FUNCTION_BLOCK FB_AlarmDelay
VAR_INPUT
	msec				: INT;
	alarmState			: BOOL;
	alarmResetTimer		: BOOL;
END_VAR
VAR_OUTPUT
	triggerAlarmState	: BOOL;
END_VAR
VAR
	tim					: TON;
END_VAR
VAR_IN_OUT
END_VAR

tim(IN:=alarmState,PT:=INT_TO_TIME(msec));

IF alarmResetTimer THEN
	tim(IN					:= FALSE);
END_IF

IF tim.Q THEN
	triggerAlarmState		:= tim.Q;
	tim(IN					:= FALSE);
	
	RETURN;
END_IF

triggerAlarmState			:=	tim.Q;

END_FUNCTION_BLOCK

(* stored: Version 1.1.0.1, ProductVersion 3.1.4022.18
   POU FB_AlarmDelay: Id {2f673dab-9385-494b-85a6-63868ddd77dd}, SpecialFunc None *)
